// TIA Portal V18 export
TYPE "UDT_Motion_Point_IAI"
// =================================================================================
//  UDT_Recipe_Final.scl
//  Version: Final
// 
//  Description:
//  Final, definitive recipe structure based on deep code analysis.
//  - Axis names and mapping are CORRECT.
//  - Position names are simple and numeric (Position_01, Position_02, ...)
//    to provide a safe, 1-to-1 mapping with the axis driver's position array.
//    This structure can be used to build a descriptive HMI.
//  =================================================================================
//  =================================================================================
//  BASE TYPES for Motion Points
//  =================================================================================
   STRUCT
      Pos : Real;   // Target Position (um/pulse)
      Vel : Int;   // Target Velocity (mm/s or %)
   END_STRUCT;
END_TYPE
